(* PLC project Unnamed, Unknown Unnamed 1 *)
(* stored: creationDateTime 2025-12-29T08:37:37, modificationDateTime 2025-12-29T08:37:37 *)

PROGRAM main
  VAR
    Relay_Start AT %QX4.0 : BOOL;  (* Address modbus: 32 *)
    Start_State AT %QX4.1 : BOOL;  (* Address modbus: 33 *)
    Relay_Downtime AT %QX4.2 : BOOL;  (* Address modbus: 34 *)
    Downtime_State AT %QX4.3 : BOOL;  (* Address modbus: 35 *)
    Counter_Trigger AT %QX4.4 : BOOL;  (* Address modbus: 36 *)
    Reset_Counter AT %QX4.5 : BOOL;  (* Address modbus: 36 *)
    Counter_Register AT %MW10 : INT;  (* 0 = 1024 --> HR 10 = 1034 *)
  END_VAR
  VAR
    R_TRIG0 : R_TRIG;
    Pulse_Counter : BOOL;
    CTU0 : CTU;
    R_TRIG1 : R_TRIG;
    Pulse_Reset : BOOL;
  END_VAR

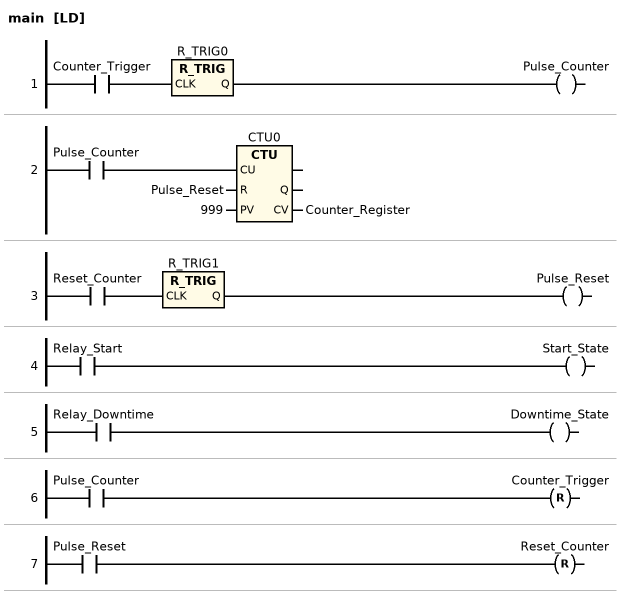
(* LD diagram, written out as Structured Text *)
Start_State := Relay_Start;
Downtime_State := Relay_Downtime;
R_TRIG0(CLK := Counter_Trigger);
Pulse_Counter := R_TRIG0.Q;
IF Pulse_Counter THEN Counter_Trigger := FALSE; END_IF;
R_TRIG1(CLK := Reset_Counter);
Pulse_Reset := R_TRIG1.Q;
IF Pulse_Reset THEN Reset_Counter := FALSE; END_IF;
CTU0(CU := Pulse_Counter, R := Pulse_Reset, PV := 999);
Counter_Register := CTU0.CV;
END_PROGRAM

CONFIGURATION Config0
  RESOURCE Res0 ON PLC
    TASK task0(INTERVAL := T#20ms, PRIORITY := 1);
    PROGRAM instance0 WITH task0 : main;
  END_RESOURCE
END_CONFIGURATION
